// TIA Portal V21 export
// export: Created 2026-09-06T18:45:55.9445964Z, ExportSetting WithDefaults, DisplayName Totally Integrated Automation Portal, DisplayVersion V21 Hotfix 1, DisplayName STEP 7 Professional, DisplayVersion V21, DisplayName STEP 7 CFC, DisplayVersion V21, DisplayName STEP 7 Safety, DisplayVersion V21, DisplayName Tech WebApplication, DisplayVersion V21, DisplayName WinCC Basic/Comfort/Advanced, DisplayVersion V21, DisplayName SIMATIC Visualization Architect, DisplayVersion V21, DisplayName WinCC Unified, DisplayVersion V21, DisplayName SIMATIC Visualization Architect, DisplayVersion V21
VAR_GLOBAL   // PLC tag table "Entradas_Expansao2_SM1221"
   M1_S4 AT %I4.0 : Bool;   // Grupo Motor M1 (Tapete 1) - Sensor S4 de Posicao / Presenca
   M1_S5 AT %I4.1 : Bool;   // Grupo Motor M1 (Tapete 1) - Sensor S5 de Posicao / Presenca
   M1_S6 AT %I4.2 : Bool;   // Grupo Motor M1 (Tapete 1) - Sensor S6 de Posicao / Presenca
   M2_S7 AT %I4.3 : Bool;   // Grupo Motor M2 (Tapete 2) - Sensor S7 de Posicao / Presenca
   M2_S8 AT %I4.4 : Bool;   // Grupo Motor M2 (Tapete 2) - Sensor S8 de Posicao / Presenca
   M2_S9 AT %I4.5 : Bool;   // Grupo Motor M2 (Tapete 2) - Sensor S9 de Posicao / Presenca
   M3_S10 AT %I4.6 : Bool;   // Grupo Motor M3 (Tapete 3) - Sensor S10 de Posicao / Presenca
   M3_S11 AT %I4.7 : Bool;   // Grupo Motor M3 (Tapete 3) - Sensor S11 de Posicao / Presenca
   M3_S12 AT %I5.0 : Bool;   // Grupo Motor M3 (Tapete 3) - Sensor S12 de Posicao / Presenca
   M4_S13 AT %I5.1 : Bool;   // Grupo Motor M4 (Tapete 4) - Sensor S13 de Posicao / Presenca
   M4_S14 AT %I5.2 : Bool;   // Grupo Motor M4 (Tapete 4) - Sensor S14 de Posicao / Presenca
   M4_S15 AT %I5.3 : Bool;   // Grupo Motor M4 (Tapete 4) - Sensor S15 de Posicao / Presenca
   M5_S16 AT %I5.4 : Bool;   // Grupo Motor M5 (Tapete 5) - Sensor S16 de Posicao / Presenca
   M5_S17 AT %I5.5 : Bool;   // Grupo Motor M5 (Tapete 5) - Sensor S17 de Posicao / Presenca
   M5_S18 AT %I5.6 : Bool;   // Grupo Motor M5 (Tapete 5) - Sensor S18 de Posicao / Presenca
   M5_S19 AT %I5.7 : Bool;   // Grupo Motor M5 (Tapete 5) - Sensor S19 de Posicao / Presenca
END_VAR
